// SIMATIC S7-200 project (STEP 7-Micro/WIN), CPU 221 REL 01.10

SYMBOL_TABLE USER1
Run              Q0.0
Dir              Q0.1
S1               I0.3
S2               I0.4
S3               I0.5
PB1              I0.0
PB2              I0.1
PB3              I0.2
END_SYMBOL_TABLE

ORGANIZATION_BLOCK MAIN:OB1
TITLE=Elevator 
BEGIN
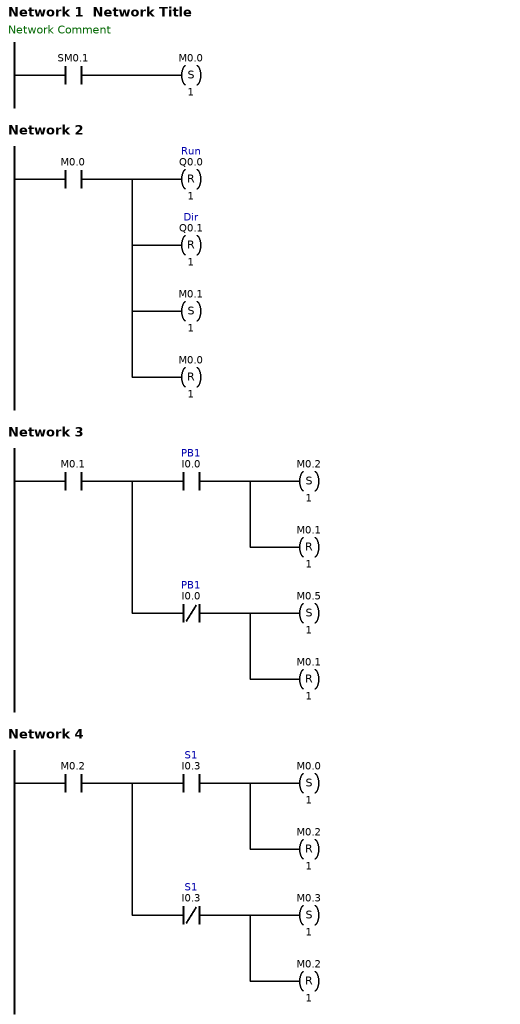
Network 1 // Network Title
// Network Comment
LD     SM0.1
S      M0.0, 1
Network 2
LD     M0.0
R      Run:Q0.0, 1
R      Dir:Q0.1, 1
S      M0.1, 1
R      M0.0, 1
Network 3
LD     M0.1
LPS
A      PB1:I0.0
S      M0.2, 1
R      M0.1, 1
LPP
AN     PB1:I0.0
S      M0.5, 1
R      M0.1, 1
Network 4
LD     M0.2
LPS
A      S1:I0.3
S      M0.0, 1
R      M0.2, 1
LPP
AN     S1:I0.3
S      M0.3, 1
R      M0.2, 1
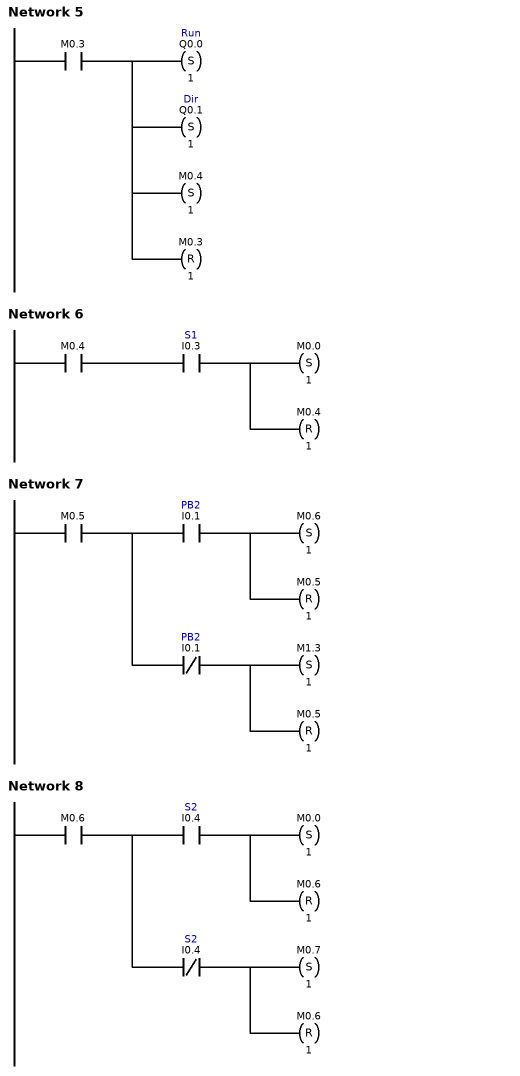
Network 5
LD     M0.3
S      Run:Q0.0, 1
S      Dir:Q0.1, 1
S      M0.4, 1
R      M0.3, 1
Network 6
LD     M0.4
A      S1:I0.3
S      M0.0, 1
R      M0.4, 1
Network 7
LD     M0.5
LPS
A      PB2:I0.1
S      M0.6, 1
R      M0.5, 1
LPP
AN     PB2:I0.1
S      M1.3, 1
R      M0.5, 1
Network 8
LD     M0.6
LPS
A      S2:I0.4
S      M0.0, 1
R      M0.6, 1
LPP
AN     S2:I0.4
S      M0.7, 1
R      M0.6, 1
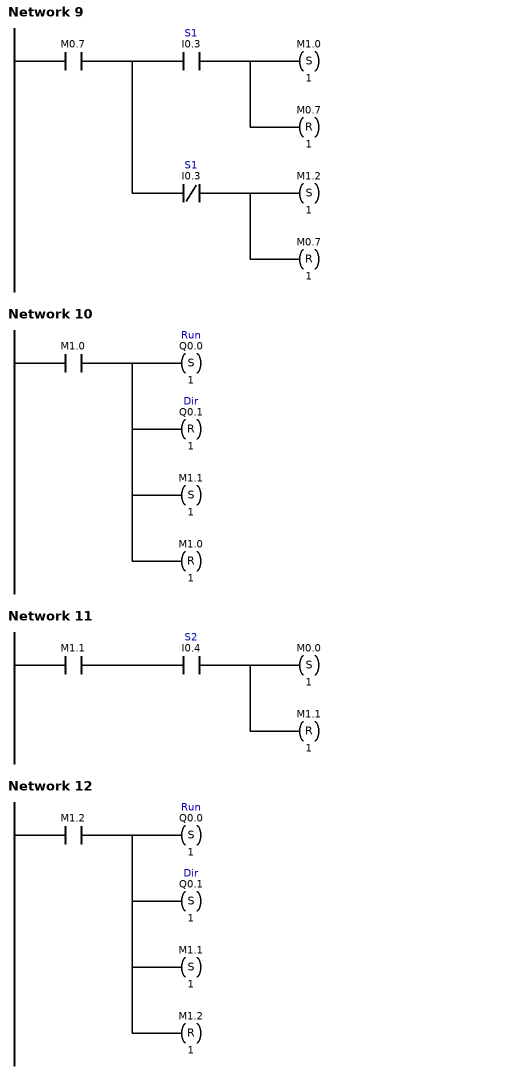
Network 9
LD     M0.7
LPS
A      S1:I0.3
S      M1.0, 1
R      M0.7, 1
LPP
AN     S1:I0.3
S      M1.2, 1
R      M0.7, 1
Network 10
LD     M1.0
S      Run:Q0.0, 1
R      Dir:Q0.1, 1
S      M1.1, 1
R      M1.0, 1
Network 11
// (network saved uncompiled; LAD cells follow)
// row 0: c0 -| |- M1.1  c1 -| |- S2:I0.4 v  c2 -(S) M0.0, 1
// row 1: c1 ^  c2 -(R) M1.1, 1
Network 12
LD     M1.2
S      Run:Q0.0, 1
S      Dir:Q0.1, 1
S      M1.1, 1
R      M1.2, 1
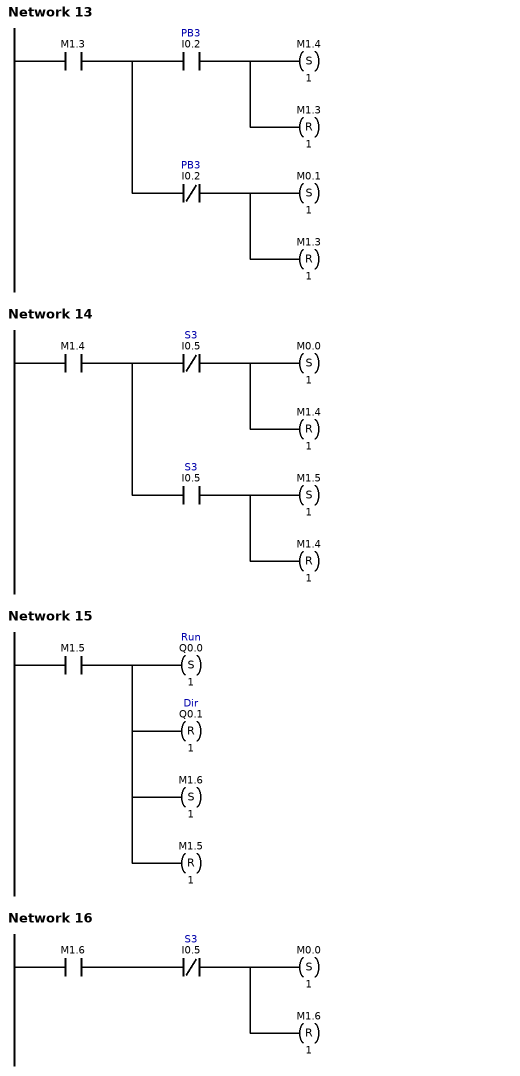
Network 13
LD     M1.3
LPS
A      PB3:I0.2
S      M1.4, 1
R      M1.3, 1
LPP
AN     PB3:I0.2
S      M0.1, 1
R      M1.3, 1
Network 14
LD     M1.4
LPS
AN     S3:I0.5
S      M0.0, 1
R      M1.4, 1
LPP
A      S3:I0.5
S      M1.5, 1
R      M1.4, 1
Network 15
LD     M1.5
S      Run:Q0.0, 1
R      Dir:Q0.1, 1
S      M1.6, 1
R      M1.5, 1
Network 16
LD     M1.6
AN     S3:I0.5
S      M0.0, 1
R      M1.6, 1
END_ORGANIZATION_BLOCK
